// TIA Portal V18 export
FUNCTION "FC_AQ" : Void   // FC10, STL
{ S7_Optimized_Access := 'TRUE' }
VERSION : 0.1
// stored: AutoNumber true, UDAEnableTagReadback false
BEGIN

NETWORK
TITLE = 

      CALL  "FC_AnalogOutCoverter"
      ( in_AnalogData  := "DB_AQ".outa_BaseAxis,
        in_NormMax     := 180.0,
        in_NormMin     := -180.0,
        out_AnalogData := "outa_BaseAxis"
      );

      CALL  "FC_AnalogOutCoverter"
      ( in_AnalogData  := "DB_AQ".outa_Arm1Axis,
        in_NormMax     := 180.0,
        in_NormMin     := -180.0,
        out_AnalogData := "outa_Arm1Axis"
      );

      CALL  "FC_AnalogOutCoverter"
      ( in_AnalogData  := "DB_AQ".outa_Arm2Axis,
        in_NormMax     := 180.0,
        in_NormMin     := -180.0,
        out_AnalogData := "outa_Arm2Axis"
      );

      CALL  "FC_AnalogOutCoverter"
      ( in_AnalogData  := "DB_AQ".outa_Arm3Axis,
        in_NormMax     := 180.0,
        in_NormMin     := -180.0,
        out_AnalogData := "outa_Arm3Axis"
      );

      CALL  "FC_AnalogOutCoverter"
      ( in_AnalogData  := "DB_AQ".outa_ToolAxis,
        in_NormMax     := 180.0,
        in_NormMin     := -180.0,
        out_AnalogData := "outa_ToolAxis"
      );

      CALL  "FC_AnalogOutCoverter"
      ( in_AnalogData  := "DB_AQ".outa_BaseSpeed,
        in_NormMax     := 180.0,
        in_NormMin     := -180.0,
        out_AnalogData := "outa_BaseSpeed"
      );

      CALL  "FC_AnalogOutCoverter"
      ( in_AnalogData  := "DB_AQ".outa_Arm1Speed,
        in_NormMax     := 180.0,
        in_NormMin     := -180.0,
        out_AnalogData := "outa_Arm1Speed"
      );

      CALL  "FC_AnalogOutCoverter"
      ( in_AnalogData  := "DB_AQ".outa_Arm2Speed,
        in_NormMax     := 180.0,
        in_NormMin     := -180.0,
        out_AnalogData := "outa_Arm2Speed"
      );

      CALL  "FC_AnalogOutCoverter"
      ( in_AnalogData  := "DB_AQ".outa_Arm3Speed,
        in_NormMax     := 180.0,
        in_NormMin     := -180.0,
        out_AnalogData := "outa_Arm3Speed"
      );

      CALL  "FC_AnalogOutCoverter"
      ( in_AnalogData  := "DB_AQ".outa_ToolSpeed,
        in_NormMax     := 180.0,
        in_NormMin     := -180.0,
        out_AnalogData := "outa_ToolSpeed"
      );

      CALL  "FC_AnalogOutCoverter"
      ( in_AnalogData  := "DB_AQ".outa_10,
        in_NormMax     := 0.0,
        in_NormMin     := 0.0,
        out_AnalogData := "outa_10"
      );

      CALL  "FC_AnalogOutCoverter"
      ( in_AnalogData  := "DB_AQ".outa_11,
        in_NormMax     := 0.0,
        in_NormMin     := 0.0,
        out_AnalogData := "outa_11"
      );

      CALL  "FC_AnalogOutCoverter"
      ( in_AnalogData  := "DB_AQ".outa_HorizontalAxis,
        in_NormMax     := 9.5,
        in_NormMin     := 0.0,
        out_AnalogData := "outa_HorizontalAxis"
      );

      CALL  "FC_AnalogOutCoverter"
      ( in_AnalogData  := "DB_AQ".outa_VerticalAxis,
        in_NormMax     := 5.0,
        in_NormMin     := 0.0,
        out_AnalogData := "outa_VerticalAxis"
      );





END_FUNCTION
